// TIA Portal V16 export
// export: Created 2024-12-03T15:41:39.4238753Z, ExportSetting WithDefaults, DisplayName Totally Integrated Automation Portal, DisplayVersion V16 Update 6, DisplayName TIA Portal Version Control Interface, DisplayVersion V16 Update 2, DisplayName TIA Portal Openness, DisplayVersion V16 Update 6, DisplayName TIA Portal Teamcenter Gateway, DisplayVersion V16, DisplayName SINAMICS Startdrive Advanced, DisplayVersion V16 Update 5, DisplayName SINAMICS Startdrive G130, G150, S120, S150, SINAMICS MV, S210, DisplayVersion V16 Update 5, DisplayName SINAMICS Startdrive G110M, G120, G120C, G120D, G120P, G115D, DisplayVersion V16 Update 5, DisplayName STEP 7 Professional, DisplayVersion V16 Update 6, DisplayName STEP 7 Safety, DisplayVersion V16, DisplayName WinCC Advanced / Unified PC, DisplayVersion V16 Update 6
FUNCTION_BLOCK "OutputsController_Scanners_FB"   // FB2, SCL
{ S7_Optimized_Access := 'TRUE' }
VERSION : 0.1
// stored: AutoNumber true, IsIECCheckEnabled false, IsRetainMemResEnabled false, MemoryReserve 100, SetENOAutomatically false, UDAEnableTagReadback false
   VAR
      SCAN_100 : "EC_Cognex_Dataman_Single_FB";
   END_VAR
BEGIN
   REGION SCAN_100

       #SCAN_100(I_HwId:="SCAN_100~Acquisition_Status_1",
                 I_Result := "I_Scan_100_ResultData",
                 I_ResultStatus := "I_Scan_100_ResultStatus",
                 I_Status := "I_Scan_100_TriggerStatus",
                 O_Control => "Q_Scan_100_ResultControl",
                 O_Trigger => "Q_Scan_100_TriggerControl",
                 IO_Scanner := "Scanners_DB".SCAN_100);

   END_REGION
END_FUNCTION_BLOCK
